Fanuc KAREL source: kt00214.KL

-- PROVISIONAL review KL for V770-1; original PC SHA256 6110106eb0b20c976ce11216f9b2b1c73c2eb6a65ee10e452b8fa7167ff8d211
-- Incomplete behavior may be omitted. Consult companion uncertainty JSON. Do not deploy.
PROGRAM KT00214
%NOLOCKGROUP
VAR
  OUT : INTEGER
-- UNRESOLVED_DECL Y1 type=002018
-- UNRESOLVED_DECL Y2 type=002018
BEGIN
  -- UNRESOLVED_PC offsets 5-19; opcodes 2E,22,9D,33,B2
  -- UNRESOLVED_PC offsets 24-38; opcodes 2E,22,9D,33,B2
  -- UNRESOLVED_PC offsets 43-57; opcodes 2E,22,9D,33,B2
  -- UNRESOLVED_PC offsets 62-76; opcodes 2E,22,9D,33,B2
  -- UNRESOLVED_PC offsets 81-106; opcodes 22,9D,33,B1,22,9D,33,B1,46,23
  -- UNRESOLVED_PC offsets 111-115; opcodes 7F
END KT00214
